Universal Robots PolyScope program: Start Heating Welder.urp

Program Start Heating Welder (installation=robot3 directory=/programs/UPF createdIn=5.14.5 lastSavedIn=5.21.2 robotSerialNumber=20256802612)
Calibrated DH parameters: a=[-0.000042, -0.384711, -0.675257, 0.000053, -0.000026, 0]; d=[0.236319, 419.71573, -259.410189, -160.105167, 0.159217, 0.154051]; alpha=[1.570689, 0.001837, -0.001695, 1.571673, -1.570506, 0]; deltaTheta=[0, 1.107921, -1.49058, 0.382655, 0.000001, 0]
InitVariablesNode
Robot Program (runOnlyOnce=true)
  HwResp := "placeholder"
  URCap WireTank Serial (WireTank Serial, WireTank, LLC) dataModel(Command=[252,72,49], NODE_TITLE=Serial Bridge uH1, byte_array=true, OUTPUT_ENTRY=Static, QUERY=false, Variable(key=OUTPUT_VARIABLE, variable=HwResp))
  ''
  ''
  Folder Folder1
    URCap WireTank Serial (WireTank Serial, WireTank, LLC) dataModel(NODE_TITLE=Serial Bridge uh?, Command=[252,104,63], OUTPUT_ENTRY=Static, QUERY=true, byte_array=true, Variable(key=OUTPUT_VARIABLE, variable(name=purge)))
    target := [252,72,49]
    resp := [1,2,3]
    URCap WireTank Serial (WireTank Serial, WireTank, LLC) dataModel(Command=[252,72,49], NODE_TITLE=Serial Bridge uH1, byte_array=true, QUERY=true, OUTPUT_ENTRY=Static, Variable(key=OUTPUT_VARIABLE, variable=resp))
    If resp≠target
      Popup Message (haltProgram=false message=could not confirm that heating started. check connection.  inputType=Text)
  SuppressedNode
    Wait Sleep waitTime=5
  SuppressedNode
    Popup Message (haltProgram=false message=heating started. push to stop inputType=Text)
  SuppressedNode
    URCap WireTank Serial (WireTank Serial, WireTank, LLC) dataModel(NODE_TITLE=Serial Bridge uh?, byte_array=true, Command=[252,104,63], OUTPUT_ENTRY=Static, QUERY=true, Variable(key=OUTPUT_VARIABLE, variable=HwResp))
  SuppressedNode
    Popup Message (haltProgram=false inputType=Variable) variable=HwResp
  SuppressedNode
    Wait Sleep waitTime=20
  SuppressedNode
    URCap WireTank Serial (WireTank Serial, WireTank, LLC) dataModel(byte_array=true, Command=[252,72,48], NODE_TITLE=Serial Bridge uH0, QUERY=false, OUTPUT_ENTRY=Static, Variable(key=OUTPUT_VARIABLE, variable=HwResp))
  SuppressedNode
    Popup Message (haltProgram=false message=heating stopped. push to start inputType=Text)
  'set the temp reader to high voltage (off) when program is running and low volt (on) when program not running'
  Script: set_runstate_standard_digital_output_to_value(2,3)
  'set 5V power to munsch powerbox to high (on) when a program is started and low on unscheduled stop'
  Script: set_runstate_standard_digital_output_to_value(1,5)
